(* IEC 61131-3 sources: ArfBotOS/Codesys-4/ArfBotOS.fbsdev/Application.iecapp^/POU/_10_Robot.prg.st^/public, 1 file *)

(* ---- M_Init.meth.st ---- *)
METHOD PUBLIC M_Init : BOOL
VAR_INPUT
	DefaultParameters: BOOL;
END_VAR

IF DefaultParameters THEN
	PersistentVars.Flags[GVL_App.INIT_DRV_IDX].Value := FALSE;
END_IF
InitializeDrives := TRUE;
END_METHOD
